FUNCTION ACVoltageCheck : BOOL
VAR_INPUT
	IN			: REAL;
END_VAR
VAR
	r_min		: REAL;
	r_max		: REAL;
END_VAR

r_min:= settings.GridParams.r_GridVoltageMin - 10;
r_max:= settings.GridParams.r_GridVoltageMax;

ACVoltageCheck := LIMIT(r_min, IN, r_max) = IN;

END_FUNCTION

(* stored: Version 1.1.0.1, ProductVersion 3.1.4026.18
   POU ACVoltageCheck: Id {95b74ab9-4c10-483b-99cc-5fc7d646e6d6}, SpecialFunc None *)
